FUNCTION_BLOCK FB_LamparaIntermitente_LD
VAR_INPUT
    TiempoParpadeo: REAL := 0.5;
END_VAR
VAR_OUTPUT
END_VAR
VAR
    Temporizador: TON;
    
    Resultado: REAL;
    Tiempo: TIME;

    Lampara AT %Q*: BOOL;
END_VAR

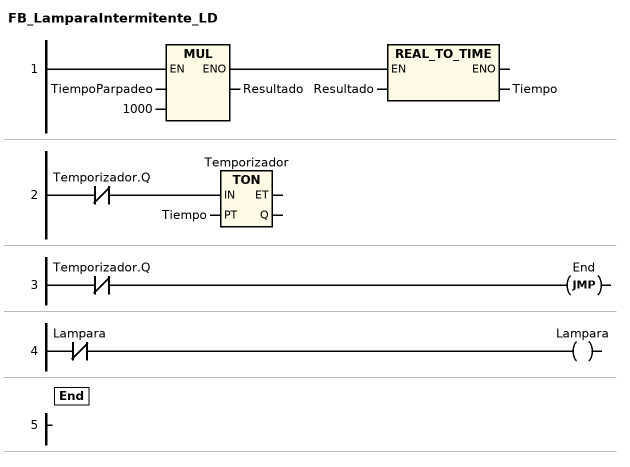
// NETWORK 1
Resultado := TiempoParpadeo * 1000;
Tiempo := REAL_TO_TIME(Resultado);

// NETWORK 2
Temporizador(IN := NOT Temporizador.Q, PT := Tiempo); // TON

// NETWORK 3
IF NOT Temporizador.Q THEN JMP End; END_IF

// NETWORK 4
Lampara := NOT Lampara;

// NETWORK 5
End: ;

END_FUNCTION_BLOCK

(* stored: Version 1.1.0.1, ProductVersion 3.1.4024.15
   POU FB_LamparaIntermitente_LD: Id {f6aef7a8-d061-4967-b273-6567cb4a7d3a}, SpecialFunc None *)
